// TIA Portal V18 export
DATA_BLOCK "Timer"   // DB59999
{ S7_Optimized_Access := 'FALSE' }
VERSION : 0.1
// stored: AutoNumber false, DBAccessibleFromOPCUA true, IsOnlyStoredInLoadMemory false, IsWriteProtectedInAS false
   VAR
      x1SecRisingEdge : Bool;   // Одноразовий ымпуьс 1сек
      x1SecPrevClock : Bool;   // Попередный стан цикоу
      x1SecFired : Bool;   // Вже вiдпрацьовано?
   END_VAR
BEGIN
END_DATA_BLOCK
